% RSLogix 500 project DIGITAL_FILLING_STATION.RSS, saved by version 8.30.00.16 %
PROJECT "PROC1"    % processor: Bul.1763 MicroLogix 1100 Series B %

PROGRAM FILES
  LAD 2 "MAIN"  4 rungs
  LAD 3 "IO"  8 rungs
  LAD 4 "CYCLES"  5 rungs
  LAD 5 "CONTROLS"  6 rungs

DATA FILES
  O0 OUTPUT  4 elements
  I1 INPUT  6 elements
  S2 STATUS  66 elements
  B3 BINARY  1 elements
  T4 TIMER  1 elements
  C5 COUNTER  1 elements
  R6 CONTROL  1 elements
  N7 INTEGER  1 elements
  F8 FLOAT  1 elements

LADDER 2 "MAIN"
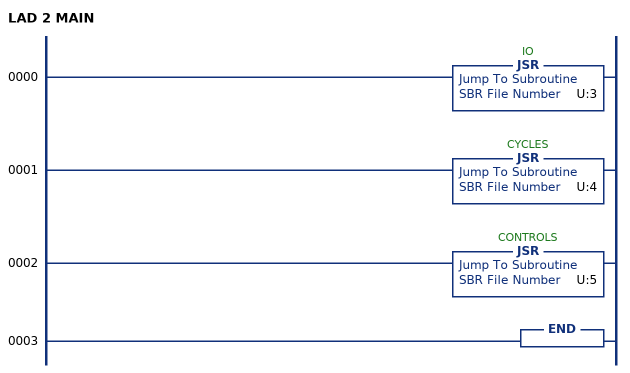
% Rung: 0 %
SOR JSR U:3 EOR
%   U:3  "IO" %
% Rung: 1 %
SOR JSR U:4 EOR
%   U:4  "CYCLES" %
% Rung: 2 %
SOR JSR U:5 EOR
%   U:5  "CONTROLS" %
% Rung: 3 %
SOR END EOR

LADDER 3 "IO"
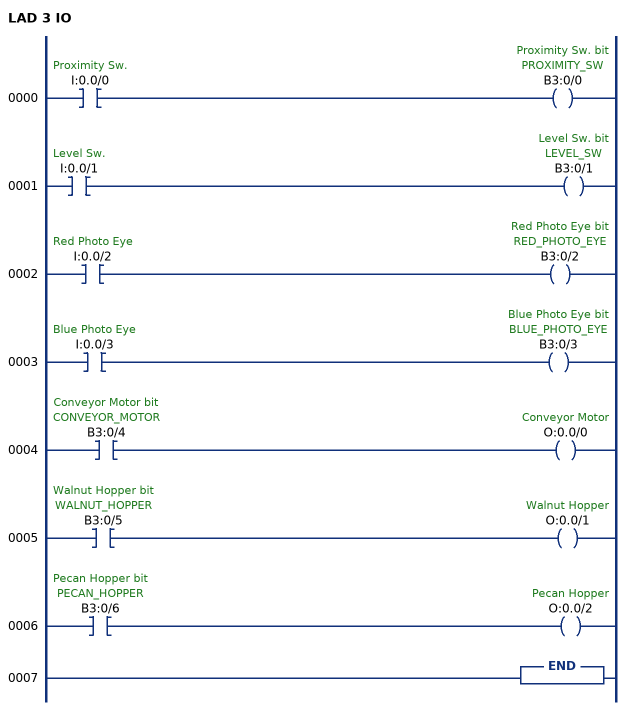
% Rung: 0 %
SOR XIC I:0.0/0 OTE B3:0/0 EOR
%   I:0.0/0  "Proximity Sw." %
%   B3:0/0  PROXIMITY_SW  "Proximity Sw. bit" %
% Rung: 1 %
SOR XIC I:0.0/1 OTE B3:0/1 EOR
%   I:0.0/1  "Level Sw." %
%   B3:0/1  LEVEL_SW  "Level Sw. bit" %
% Rung: 2 %
SOR XIC I:0.0/2 OTE B3:0/2 EOR
%   I:0.0/2  "Red Photo Eye" %
%   B3:0/2  RED_PHOTO_EYE  "Red Photo Eye bit" %
% Rung: 3 %
SOR XIC I:0.0/3 OTE B3:0/3 EOR
%   I:0.0/3  "Blue Photo Eye" %
%   B3:0/3  BLUE_PHOTO_EYE  "Blue Photo Eye bit" %
% Rung: 4 %
SOR XIC B3:0/4 OTE O:0.0/0 EOR
%   B3:0/4  CONVEYOR_MOTOR  "Conveyor Motor bit" %
%   O:0.0/0  "Conveyor Motor" %
% Rung: 5 %
SOR XIC B3:0/5 OTE O:0.0/1 EOR
%   B3:0/5  WALNUT_HOPPER  "Walnut Hopper bit" %
%   O:0.0/1  "Walnut Hopper" %
% Rung: 6 %
SOR XIC B3:0/6 OTE O:0.0/2 EOR
%   B3:0/6  PECAN_HOPPER  "Pecan Hopper bit" %
%   O:0.0/2  "Pecan Hopper" %
% Rung: 7 %
SOR END EOR

LADDER 4 "CYCLES"
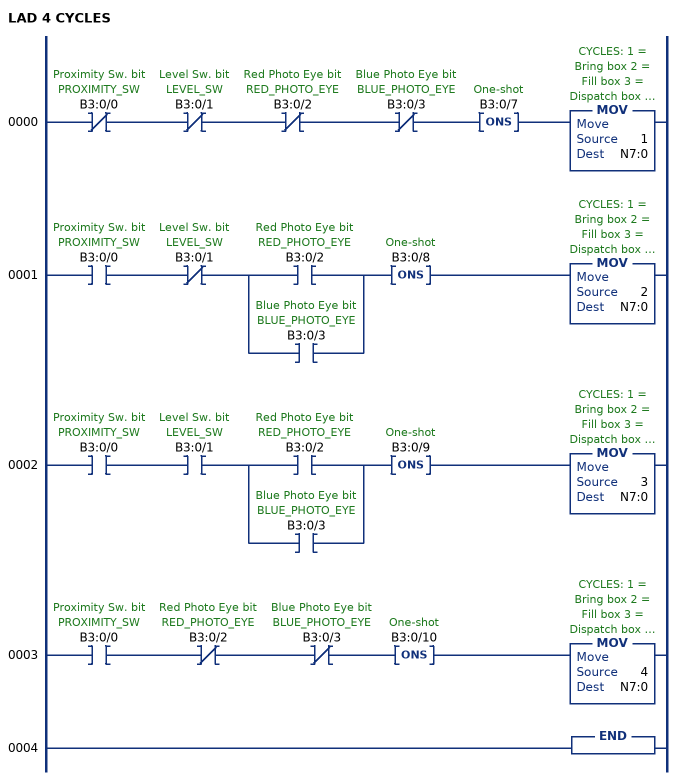
% Rung: 0 %
SOR XIO B3:0/0 XIO B3:0/1 XIO B3:0/2 XIO B3:0/3 ONS B3:0/7 MOV 1 N7:0 EOR
%   B3:0/0  PROXIMITY_SW  "Proximity Sw. bit" %
%   B3:0/1  LEVEL_SW  "Level Sw. bit" %
%   B3:0/2  RED_PHOTO_EYE  "Red Photo Eye bit" %
%   B3:0/3  BLUE_PHOTO_EYE  "Blue Photo Eye bit" %
%   B3:0/7  "One-shot" %
%   N7:0  N7  "CYCLES: 1 = Bring box 2 = Fill box 3 = Dispatch box 4 = Label undetected" %
% Rung: 1 %
SOR XIC B3:0/0 XIO B3:0/1 BST XIC B3:0/2 NXB XIC B3:0/3 BND ONS B3:0/8 MOV 2 N7:0 EOR
%   B3:0/0  PROXIMITY_SW  "Proximity Sw. bit" %
%   B3:0/1  LEVEL_SW  "Level Sw. bit" %
%   B3:0/2  RED_PHOTO_EYE  "Red Photo Eye bit" %
%   B3:0/3  BLUE_PHOTO_EYE  "Blue Photo Eye bit" %
%   B3:0/8  "One-shot" %
%   N7:0  N7  "CYCLES: 1 = Bring box 2 = Fill box 3 = Dispatch box 4 = Label undetected" %
% Rung: 2 %
SOR XIC B3:0/0 XIC B3:0/1 BST XIC B3:0/2 NXB XIC B3:0/3 BND ONS B3:0/9 MOV 3 N7:0 EOR
%   B3:0/0  PROXIMITY_SW  "Proximity Sw. bit" %
%   B3:0/1  LEVEL_SW  "Level Sw. bit" %
%   B3:0/2  RED_PHOTO_EYE  "Red Photo Eye bit" %
%   B3:0/3  BLUE_PHOTO_EYE  "Blue Photo Eye bit" %
%   B3:0/9  "One-shot" %
%   N7:0  N7  "CYCLES: 1 = Bring box 2 = Fill box 3 = Dispatch box 4 = Label undetected" %
% Rung: 3 %
SOR XIC B3:0/0 XIO B3:0/2 XIO B3:0/3 ONS B3:0/10 MOV 4 N7:0 EOR
%   B3:0/0  PROXIMITY_SW  "Proximity Sw. bit" %
%   B3:0/2  RED_PHOTO_EYE  "Red Photo Eye bit" %
%   B3:0/3  BLUE_PHOTO_EYE  "Blue Photo Eye bit" %
%   B3:0/10  "One-shot" %
%   N7:0  N7  "CYCLES: 1 = Bring box 2 = Fill box 3 = Dispatch box 4 = Label undetected" %
% Rung: 4 %
SOR END EOR

LADDER 5 "CONTROLS"
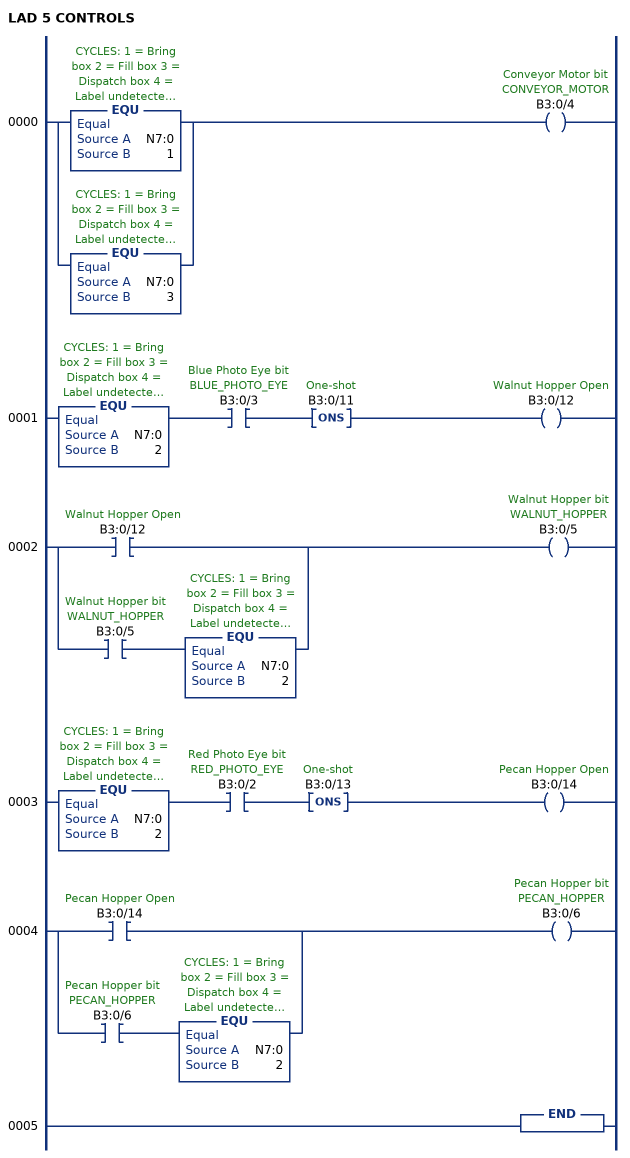
% Rung: 0 %
SOR BST EQU N7:0 1 NXB EQU N7:0 3 BND OTE B3:0/4 EOR
%   N7:0  N7  "CYCLES: 1 = Bring box 2 = Fill box 3 = Dispatch box 4 = Label undetected" %
%   B3:0/4  CONVEYOR_MOTOR  "Conveyor Motor bit" %
% Rung: 1 %
SOR EQU N7:0 2 XIC B3:0/3 ONS B3:0/11 OTE B3:0/12 EOR
%   N7:0  N7  "CYCLES: 1 = Bring box 2 = Fill box 3 = Dispatch box 4 = Label undetected" %
%   B3:0/3  BLUE_PHOTO_EYE  "Blue Photo Eye bit" %
%   B3:0/11  "One-shot" %
%   B3:0/12  "Walnut Hopper Open" %
% Rung: 2 %
SOR BST XIC B3:0/12 NXB XIC B3:0/5 EQU N7:0 2 BND OTE B3:0/5 EOR
%   B3:0/12  "Walnut Hopper Open" %
%   B3:0/5  WALNUT_HOPPER  "Walnut Hopper bit" %
%   N7:0  N7  "CYCLES: 1 = Bring box 2 = Fill box 3 = Dispatch box 4 = Label undetected" %
% Rung: 3 %
SOR EQU N7:0 2 XIC B3:0/2 ONS B3:0/13 OTE B3:0/14 EOR
%   N7:0  N7  "CYCLES: 1 = Bring box 2 = Fill box 3 = Dispatch box 4 = Label undetected" %
%   B3:0/2  RED_PHOTO_EYE  "Red Photo Eye bit" %
%   B3:0/13  "One-shot" %
%   B3:0/14  "Pecan Hopper Open" %
% Rung: 4 %
SOR BST XIC B3:0/14 NXB XIC B3:0/6 EQU N7:0 2 BND OTE B3:0/6 EOR
%   B3:0/14  "Pecan Hopper Open" %
%   B3:0/6  PECAN_HOPPER  "Pecan Hopper bit" %
%   N7:0  N7  "CYCLES: 1 = Bring box 2 = Fill box 3 = Dispatch box 4 = Label undetected" %
% Rung: 5 %
SOR END EOR
